/// <summary>
/// Motors with one direction of rotation
/// Motoren mit einer Drehrichtung
/// </summary>
FUNCTION_BLOCK PUBLIC PAEEMotor1D EXTENDS PAEEMotorStartCtrl
VAR_INPUT
	_IRun AT %I*: BOOL;	
END_VAR
VAR_OUTPUT
	_QRun AT %Q*: BOOL;	
END_VAR
VAR
	_PAPointMatIn1 : PAPoint(THIS^);
	_PAPointMatOut1 : PAPoint(THIS^);
END_VAR

METHOD FB_init : BOOL
VAR_INPUT
	bInitRetains : BOOL; // if TRUE, the retain variables are initialized (warm start / cold start)
	bInCopyCode : BOOL;  // if TRUE, the instance afterwards gets moved into the copy code (online change)
	parent : IACComponent;
END_VAR
AddPoint(_PAPointMatIn1);
AddPoint(_PAPointMatOut1);
END_METHOD

METHOD PUBLIC HasPointReachedOffPosition : BOOL
VAR_INPUT
	point : IACPoint;
END_VAR
IF point = PAPointMatOut1 THEN
	HasPointReachedOffPosition := NOT _RunState;
ELSIF point = PAPointMatIn1 THEN
	HasPointReachedOffPosition := TRUE;
ELSE
	HasPointReachedOffPosition := FALSE;
END_IF
END_METHOD

METHOD PUBLIC HasPointReachedOnPosition : BOOL
VAR_INPUT
	point : IACPoint;
END_VAR
IF point = PAPointMatOut1 THEN
	HasPointReachedOnPosition := _RunState;
ELSIF point = PAPointMatIn1 THEN
	HasPointReachedOnPosition := TRUE;
ELSE
	HasPointReachedOnPosition := FALSE;
END_IF
END_METHOD

METHOD PUBLIC IsEnabledTurnOn : BOOL
VAR_INPUT
END_VAR
END_METHOD

METHOD PROTECTED OnMainEnter
VAR_INPUT
END_VAR
_QRun := THIS^._ReqRunState;
END_METHOD

PROPERTY PUBLIC PAPointMatIn1 : IACPoint
GET // PUBLIC
PAPointMatIn1 := _PAPointMatIn1;
END_GET
END_PROPERTY

PROPERTY PUBLIC PAPointMatOut1 : IACPoint
GET // PUBLIC
PAPointMatOut1 := _PAPointMatOut1;
END_GET
END_PROPERTY

METHOD PUBLIC TurnOn
VAR_INPUT
END_VAR
END_METHOD

END_FUNCTION_BLOCK

(* stored: Version 1.1.0.1, ProductVersion 3.1.4020.12
   POU PAEEMotor1D: Id {56c3d8a1-e003-48f1-ad8e-d32a0d33e1b8}, SpecialFunc None
   Method FB_init: Id {cbbc8d50-ad60-4cce-b5f5-08bfd68a83fa}
   Method HasPointReachedOffPosition: Id {f11c36e2-5698-4c01-ab2a-115358c8f1bd}
   Method HasPointReachedOnPosition: Id {fefdf554-209b-4e51-b8ca-46ac62d4e4dc}
   Method IsEnabledTurnOn: Id {f75bd769-5e90-46cf-8dc9-a6366ef114f8}
   Method OnMainEnter: Id {4b20fc4b-f5ff-45d6-ae5d-fb5a5f099dc3}
   Property PAPointMatIn1: Id {3d82a3b8-cf7c-424d-b1b2-7bbafa777e7c}
   Get Get: Id {4dae7783-f586-440e-9b96-ae711b8cd648}
   Property PAPointMatOut1: Id {880387f7-3a50-4d6e-9c26-49c5bd747146}
   Get Get: Id {f3554bd4-ab10-47ab-bdf7-c3e5120040b9}
   Method TurnOn: Id {9e881d70-a14c-4e76-a3e6-9ee77c00e785} *)
